// TIA Portal V18 export
// export: Created 2026-03-12T16:04:34.5404943Z, ExportSetting WithDefaults, DisplayName Totally Integrated Automation Portal, DisplayVersion V18 Update 5, DisplayName TIA Portal Openness, DisplayVersion V18 Update 5, DisplayName TIA Portal Version Control Interface, DisplayVersion V18, DisplayName SINAMICS Startdrive Advanced, DisplayVersion V18, DisplayName SINAMICS Startdrive G130, G150, S120, S150, SINAMICS MV, S210, DisplayVersion V18, DisplayName SINAMICS Startdrive G110M, G120, G120C, G120D, G120P, G115D, DisplayVersion V18, DisplayName STEP 7 Professional, DisplayVersion V18 Update 5, DisplayName STEP 7 Safety, DisplayVersion V18, DisplayName WinCC Professional, DisplayVersion V18 Update 5
FUNCTION_BLOCK "SINA_SPEED_TLG20"   // FB38003, SCL
TITLE = Speed control S7 to SINAMICS using Standardtelegram 20
{ S7_Optimized_Access := 'TRUE' }
AUTHOR : SIEMENS
FAMILY : DRIVES
NAME : SINA_SPD_TLG20
VERSION : 1.0
// The function block SINA_SPEED_TLG20 controls a SINAMICS drive using standard telegram 20
// stored: AutoNumber false, IsIECCheckEnabled false, IsRetainMemResEnabled false, MemoryReserve 100, SetENOAutomatically false, UDAEnableTagReadback false
   VAR_INPUT
      enableAxis : Bool;   // 0 -> 1 = Enable the drive (OFF2 / OFF 3 are 1 in default status) (OFF1 = 0->1)
      ackError : Bool;   // 0 -> 1 = Acknowledge drive error
      speedSp : Real;   // Speed setpoint [rpm]
      selectCDS : USInt;   // Selection of the Command Data Set (0 = CDS0, 1 = CDS1)
      refSpeed : Real;   // Reference speed [p2000] in [rpm]
      refCurrent : Real;   // Reference current [p2002] in [Aeff]
      refTorque : Real;   // Reference torque [p2003] in [Nm]
      refPower : Real;   // Reference power [r2005] in [kW]
      configAxis : Word := 16#003F;   // binary programmed input to control all functions in the telegram without its own function block input
      HWIDSTW : HW_IO;   // Hardware Identifer set point slot
      HWIDZSW : HW_IO;   // Hardware Identifer actual value slot
   END_VAR
   VAR_OUTPUT
      axisEnabled : Bool;   // 1 = Drive is enabled
      lockout : Bool;   // 1 = Drive lockout active
      actCDS : USInt;   // Active Command Data Set (0 = CDS0, 1 = CDS1)
      actSpeed : Real;   // Smoothed actual speed in [1/min]
      actCurrent : Real;   // Smoothed current actual in [Arms]
      actTorque : Real;   // Actual smoothed torque in [Nm]
      actPower : Real;   // Actual smoothed active power in [kW]
      faultVIKNAMUR : Word;   // Fault word according to the VIK-NAMUR defintion
      error : Bool;   // 1 = Error (FB and Infeed)
      status : Int;   // Status output (7002 = FB in operation; 7xxx = warning; 8xxx = error description - read the manual)
      diagId : Int;   // Error codes of the system function blocks DPWR / DPRD_DAT
   END_VAR
   VAR_TEMP
      tempSpeed : Real;   // Speed setpoint in percent
      tempRefValueInvalid : Bool;   // At least one reference value is 0 or < 0
      tempSendBuf : Array[0..1] of Word;   // Send buffer
      tempRecvBuf : Array[0..5] of Word;   // Receive buffer
   END_VAR
   VAR CONSTANT
      NORMALIZATION_VALUE : Int := 16#4000;   // Used to calculate the Real values
      MAX_INT : Int := 16#7FFF;
      MIN_INT : Int := 16#8000;
      REF_CURRRENT_INVALID : Int := 16#7010;   // RefCurrent input is 0 or < 0
      REF_TORQUE_INVALID : Int := 16#7011;   // RefTorque input is 0 or < 0
      REF_POWER_INVALID : Int := 16#7012;   // RefPower input is 0 or < 0
      REF_VALUES_INVALID : Int := 16#7013;   // Multiple reference values are 0 or < 0
      NO_ERROR : Int := 16#7002;   // No error
      ERROR_REF_SPEED_INVALID : Int := 16#8001;   // RefSpeed input is 0 or < 0
      ERROR_INVALID_CDS : Int := 16#8002;   // Invalid Command Data Set selected
      ERROR_DRIVE : Int := 16#8401;   // Drive error
      ERROR_LOCKOUT : Int := 16#8402;   // Drive lockout
      ERROR_DPREAD : Int := 16#8600;   // DPRD_DAT returned an error
      ERROR_DPWRITE : Int := 16#8601;   // DPWR_DAT returned an error
      ERROR_FAULT_WORD : Int := 16#8700;   // faultVIKNAMUR is not 0
      STW1 : USInt := 0;
      ZSW1 : USInt := 0;
      NSOLL_A : USInt := 1;
   END_VAR
BEGIN
   //=============================================================================
   //SIEMENS AG
   //(c)Copyright 2019 All Rights Reserved
   //-----------------------------------------------------------------------------
   // Library:       LSINAExt
   // Tested with:   SIMATIC S7 CPU 1513-1 PN V2.5
   // Engineering:   TIA Portal V15
   // Restrictions:  -
   // Requirements:  S7-1200 / S7-1500
   // Functionality: cyclic communication between a SINAMICS a PLC.
   //                If in HWConfig standard telegram 20 are projected 2 PZD-words are exchanged
   //                in every bus cycle.
   //                The parametrisation of these words is described in the manual of the
   //                SINAMICS
   //-----------------------------------------------------------------------------
   //Change log table:
   //Version  Date       Expert in charge Changes applied
   //01.00.00 11.02.2019 (AS) First released version
   //=============================================================================

   // Prepare PZD1 (STW1)
   #tempSendBuf[STW1].%X0 := #enableAxis;
   #tempSendBuf[STW1].%X7 := #ackError;
   #tempSendBuf[STW1].%X1 := #configAxis.%X0;
   #tempSendBuf[STW1].%X2 := #configAxis.%X1;
   #tempSendBuf[STW1].%X3 := #configAxis.%X2;
   #tempSendBuf[STW1].%X4 := #configAxis.%X3;
   #tempSendBuf[STW1].%X5 := #configAxis.%X4;
   #tempSendBuf[STW1].%X6 := #configAxis.%X5;
   #tempSendBuf[STW1].%X11 := #configAxis.%X6;
   #tempSendBuf[STW1].%X15 := #selectCDS = 1; // true = CDS0, false = CDS1
   #tempSendBuf[STW1].%X10 := TRUE; // control by PLC
   #tempSendBuf[STW1].%X13 := FALSE; // STW1.X13 not used in Telegram 20
   #tempSendBuf[STW1].%X14 := FALSE; // STW1.X14 not used in Telegram 20

   // Check CDS index
   IF (#selectCDS < 0)
       OR (#selectCDS > 1)
   THEN
       #error := TRUE;
       #status := #ERROR_INVALID_CDS;
       #tempSendBuf[STW1].%X0 := FALSE; // disable axis
   END_IF;

   // Speed
   IF #refSpeed > 0 THEN
       #tempSpeed := #speedSp * (#NORMALIZATION_VALUE / #refSpeed);
       // Limit REAL - Variable to INT - limits
       IF #tempSpeed > #MAX_INT
       THEN
           #tempSpeed := #MAX_INT;
       ELSIF #tempSpeed < #MIN_INT
       THEN
           #tempSpeed := #MIN_INT;
       ELSE
           ; // not needed
       END_IF;
       #tempSendBuf[NSOLL_A] := INT_TO_WORD(REAL_TO_INT(#tempSpeed));
   ELSE
       #error := TRUE;
       #status := #ERROR_REF_SPEED_INVALID;
       #tempSendBuf[NSOLL_A] := W#16#0;
   END_IF;

   // Send telegram to drive
   #diagId := DPWR_DAT(LADDR := #HWIDSTW,
                       RECORD := #tempSendBuf);

   // Error when writing the telegram
   IF #diagId <> 0 THEN
       #error := TRUE;
       #status := #ERROR_DPWRITE;

       // Reset outputs
       #actSpeed := 0.0;
       #actCurrent := 0.0;
       #actTorque := 0.0;
       #actPower := 0.0;
       #faultVIKNAMUR := W#16#0;

       RETURN;
   ELSE
       ;
   END_IF;

   // Receive telegram from drive
   #diagId := DPRD_DAT(LADDR := #HWIDZSW,
                       RECORD => #tempRecvBuf);

   // Error when reading the telegram
   IF #diagId <> 0 THEN
       #error := TRUE;
       #status := #ERROR_DPREAD;

       // Reset outputs
       #actSpeed := 0.0;
       #actCurrent := 0.0;
       #actTorque := 0.0;
       #actPower := 0.0;
       #faultVIKNAMUR := W#16#0;

       RETURN;
   ELSE
       ;
   END_IF;

   // Analyse ZSW1
   #axisEnabled := #tempRecvBuf[ZSW1].%X2;
   #lockout := #tempRecvBuf[ZSW1].%X6;
   #error := #tempRecvBuf[ZSW1].%X3 OR #tempRecvBuf[ZSW1].%X6;

   IF #tempRecvBuf[ZSW1].%X3 THEN
       #status := #ERROR_DRIVE;
   ELSIF #tempRecvBuf[ZSW1].%X6 THEN
       #status := #ERROR_LOCKOUT;
   ELSE
       #status := #NO_ERROR;
   END_IF;

   // Check CDS
   IF #tempRecvBuf[ZSW1].%X15 THEN
       #actCDS := 1;
   ELSE
       #actCDS := 0;
   END_IF;

   //IF #actCDS <> #selectCDS THEN
   //  #error := TRUE;
   //  #status := #ERROR_INVALID_CDS;
   //END_IF;

   // Actual speed
   IF (#refSpeed <= 0)
       AND #enableAxis
   THEN
       #actSpeed := 0.0;
       #error := TRUE;
       #status := #ERROR_REF_SPEED_INVALID;
   ELSE
       #actSpeed := INT_TO_REAL(WORD_TO_INT(#tempRecvBuf[1])) / (#NORMALIZATION_VALUE / #refSpeed);
   END_IF;

   // Actual current
   IF (#refCurrent <= 0)
       AND #enableAxis
       AND NOT #error
   THEN
       #actCurrent := 0.0;

       IF #tempRefValueInvalid THEN
           #status := #REF_VALUES_INVALID;
       ELSE
           #status := #REF_CURRRENT_INVALID;
           #tempRefValueInvalid := TRUE;
       END_IF;
   ELSE
       #actCurrent := INT_TO_REAL(WORD_TO_INT(#tempRecvBuf[2])) / (#NORMALIZATION_VALUE / #refCurrent);
   END_IF;

   // Actual torque
   IF (#refTorque <= 0)
       AND #enableAxis
       AND NOT #error
   THEN
       #actTorque := 0.0;

       IF #tempRefValueInvalid THEN
           #status := #REF_VALUES_INVALID;
       ELSE
           #status := #REF_TORQUE_INVALID;
           #tempRefValueInvalid := TRUE;
       END_IF;
   ELSE
       #actTorque := INT_TO_REAL(WORD_TO_INT(#tempRecvBuf[3])) / (#NORMALIZATION_VALUE / #refTorque);
   END_IF;

   // Actual active power
   IF (#refPower <= 0)
       AND #enableAxis
       AND NOT #error
   THEN
       #actPower := 0.0;

       IF #tempRefValueInvalid THEN
           #status := #REF_VALUES_INVALID;
       ELSE
           #status := #REF_POWER_INVALID;
           #tempRefValueInvalid := TRUE;
       END_IF;
   ELSE
       #actPower := INT_TO_REAL(WORD_TO_INT(#tempRecvBuf[4])) / (#NORMALIZATION_VALUE / #refPower);
   END_IF;

   // VIKNAMUR fault word
   #faultVIKNAMUR := #tempRecvBuf[5];
   IF #faultVIKNAMUR <> 16#0000 THEN
       #error := TRUE;
       #status := #ERROR_FAULT_WORD;
   ELSE
       ;
   END_IF;
END_FUNCTION_BLOCK
